(* Logix 5000 project; controller ProyectoAPM Emulate 5570 rev 30.12; software revision 30.00 *)

TASK MainTask (continuous, watchdog 500 ms) : MainProgram

MODULES
   Local : Emulate 5570 (ICP 2, rev 30.12)
      VIRTUAL_OUTPUTS : vendor 1 type 0 code 15 (ICP 4, rev 1.1, Output RPI 50 ms)
      VIRTUAL_INPUTS : vendor 1 type 0 code 15 (ICP 3, rev 1.1, Output RPI 50 ms)
END_MODULES

TYPE HOLE_POSITION :
STRUCT
   X : REAL;
   Y : REAL;
   Z : REAL;
   Z_Hole : REAL;
END_STRUCT
END_TYPE

VAR_GLOBAL   (* controller tags *)
   CNC0_CVB_RUN : BOOL;
   CNC0_CVB_SNR : BOOL;
   DRI0_AXIS_RUN : BOOL;
   DRI0_AXIS_X_AIM_POS : REAL;
   DRI0_AXIS_X_POS : REAL;
   DRI0_AXIS_X_SNR : REAL;
   DRI0_AXIS_Y_AIM_POS : REAL;
   DRI0_AXIS_Y_POS : REAL;
   DRI0_AXIS_Y_SNR : REAL;
   DRI0_AXIS_Z_AIM_POS : REAL;
   DRI0_AXIS_Z_POS : REAL;
   DRI0_AXIS_Z_SNR : REAL;
   DRI0_CVB_RUN : BOOL;
   DRI0_CVB_SNR : BOOL;
   HOLES_PER_TEMPLATE : DINT[4] := ([0] := 20, [1] := 4, [2] := 4, [3] := 4); {constant}
   Hommed : BOOL;
   MOR0_C0_BSW : BOOL;
   MOR0_C0_ESW : BOOL;
   MOR0_C0_VAL : BOOL;
   MOR0_C1_BSW : BOOL;
   MOR0_C1_ESW : BOOL;
   MOR0_C1_VAL : BOOL;
   MOR1_C0_BSW : BOOL;
   MOR1_C0_ESW : BOOL;
   MOR1_C0_VAL : BOOL;
   MOR1_C1_BSW : BOOL;
   MOR1_C1_ESW : BOOL;
   MOR1_C1_VAL : BOOL;
   PAN0_DRI0_CVB_RUN_PB : BOOL;
   PAN0_RST_PB : BOOL;
   PAN0_STP_PB : BOOL;
   PAN0_STT_PB : BOOL;
   PIN0_CVB_RUN : BOOL;
   PIN0_CVB_SNR : BOOL;
   RBT0_CNC0_CVB_RUN : BOOL;
   RBT0_CNC0_CVB_SNR : BOOL;
   RBT0_PIN0_CVB_RUN : BOOL;
   RBT0_PIN0_CVB_SNR : BOOL;
   RBT0_RST_PB : BOOL;
   RBT0_STP_PB : BOOL;
   RBT0_STT_PB : BOOL;
   RBT0_VAL_RUN : BOOL;
   RMT_CNC0_CVB_RUN : BOOL;
   S0_INIT : BOOL;
   S1_CFG : BOOL;
   S2_STBY : BOOL;
   S3_CNC0 : BOOL;
   S3_S0_RUN : BOOL;   // CNC0 Operación Normal de Cinta Transportadora
   S3_S1_STP : BOOL;   // CNC0 Parada de Cinta Transportadora
   S3_S2_STT : BOOL;   // CNC0 Arranque de Cinta Transportadora
   S3_Timer : TIMER := (PRE := 2000);
   S3_TIMER2 : TIMER := (PRE := 10);
   S4_CVB_RQ_ACK : BOOL;
   S4_PIN0 : BOOL;
   S4_S0_RUN : BOOL;   // PIN0 Operación normal de la cinta transportadora con mordazas abiertas
   S4_S1_STP : BOOL;   // PIN0 Parada de Cinta transportadora
   S4_S2_CLE : BOOL;   // PIN0 Cierre de mordazas
   S4_S3_OPN : BOOL;   // PIN0 Apertura de mordazas
   S4_S4_STT : BOOL;   // PIN0 Arranque de cinta transportadora
   S4_Timer0 : TIMER := (PRE := 1000);
   S4_Timer1 : TIMER := (PRE := 2000);
   S4_TIMER2 : TIMER := (PRE := 10);
   S5_COUNTS : INT;
   S5_CURRENT_TEMPLATE : DINT;
   S5_CVB_RQ : BOOL;
   S5_DRI0 : BOOL;
   S5_S0_BYS : BOOL;   // DRI0 Estado de bypass de pasada de primeras piezas
   S5_S1_WAIT_DONE : BOOL;
   S5_S1_WAT : BOOL;   // DRI0 Estato de espera de conteo de primeras piezas
   S5_S1_WAT_END : BOOL;
   S5_S2_RUN : BOOL;   // DRI0 Operación normal de la cinta transportadora con mordazas abiertas
   S5_S3_S0_SBY : BOOL;
   S5_S3_STP : BOOL;   // DRI0 Parada de Cinta transportadora
   S5_S4_CLE : BOOL;   // DRI0 Cierre de mordazas
   S5_S5_DRI : BOOL;   // DRI0 Taladrado
   S5_S5_S0_MOV : BOOL;
   S5_S5_S1_HLE : BOOL;
   S5_S5_S2_UP : BOOL;
   S5_S5_S3_ITR : BOOL;
   S5_S5_S4_EVL : BOOL;
   S5_S5_TIMER0 : TIMER := (PRE := 1000);
   S5_S5_TIMER1 : TIMER := (PRE := 1000);
   S5_S5_TIMER10 : TIMER := (PRE := 1000);
   S5_S5_TIMER11 : TIMER := (PRE := 1000);
   S5_S5_TIMER2 : TIMER := (PRE := 1000);
   S5_S5_TIMER3 : TIMER := (PRE := 1000);
   S5_S5_TIMER4 : TIMER := (PRE := 1000);
   S5_S5_TIMER5 : TIMER := (PRE := 1000);
   S5_S5_TIMER6 : TIMER := (PRE := 1000);
   S5_S5_TIMER7 : TIMER := (PRE := 1000);
   S5_S5_TIMER8 : TIMER := (PRE := 1000);
   S5_S5_TIMER9 : TIMER := (PRE := 1000);
   S5_S6_OPN : BOOL;   // DRI0 Apertura de Mordazas
   S5_S7_STT : BOOL;   // DRI0 Arranque de cinta transportadora durante 2 segundos
   S5_Timer0 : TIMER := (PRE := 2000);
   S5_Timer1 : TIMER := (PRE := 1000);
   S5_Timer2 : TIMER := (PRE := 2000);
   S5_TMP1_IDX : DINT;
   S5_TMP1_INIT : BOOL;
   T0 : BOOL;
   T1 : BOOL;
   T2 : BOOL;
   T3 : BOOL;
   T4 : BOOL;
   T5 : BOOL;
   TEMPLATE1_HOLES : HOLE_POSITION[20] := ([0].X := 14.178, [0].Y := 12.636, [0].Z := 15.692, [0].Z_Hole := 0.692, [1].X := 53.069, [1].Y := 19.708, [1].Z := 15.692, [1].Z_Hole := 0.692, [2].X := 14.178, [2].Y := 177.636, [2].Z := 15.692, [2].Z_Hole := 0.692, [3].X := 14.178, [3].Y := 177.636, [3].Z := 15.692, [3].Z_Hole := 0.692, [4].X := 53.069, [4].Y := 184.708, [4].Z := 15.692, [4].Z_Hole := 0.692, [5].X := 74.282, [5].Y := 205.921, [5].Z := 15.692, [5].Z_Hole := 0.692, [6].X := 14.178, [6].Y := 342.636, [6].Z := 15.692, [6].Z_Hole := 0.692, [7].X := 53.069, [7].Y := 349.708, [7].Z := 15.692, [7].Z_Hole := 0.692, [8].X := 74.282, [8].Y := 370.921, [8].Z := 15.692, [8].Z_Hole := 0.692, [9].X := 14.178, [9].Y := 507.636, [9].Z := 15.692, [9].Z_Hole := 0.692, [10].X := 53.069, [10].Y := 514.708, [10].Z := 15.692, [10].Z_Hole := 0.692, [11].X := 74.282, [11].Y := 535.921, [11].Z := 15.692, [11].Z_Hole := 0.692, [12].X := 134.945, [12].Y := 81.897, [12].Z := 15.692, [12].Z_Hole := 0.692, [13].X := 134.945, [13].Y := 95.897, [13].Z := 15.692, [13].Z_Hole := 0.692, [14].X := 134.156, [14].Y := 440.028, [14].Z := 15.692, [14].Z_Hole := 0.692,
        [15].X := 134.156, [15].Y := 454.028, [15].Z := 15.692, [15].Z_Hole := 0.692, [16].X := 342.588, [16].Y := 142.755, [16].Z := 292.792, [16].Z_Hole := 256.992, [17].X := 342.588, [17].Y := 446.594, [17].Z := 292.792, [17].Z_Hole := 256.992, [18].X := 412.588, [18].Y := 142.755, [18].Z := 292.792, [18].Z_Hole := 256.992, [19].X := 412.588, [19].Y := 446.594, [19].Z := 292.792, [19].Z_Hole := 256.992); {constant}
   TEMPLATE2_HOLES : HOLE_POSITION[4] := ([0].X := 73.196, [0].Y := 300.262, [0].Z := 15.692, [0].Z_Hole := 0.692, [1].X := 225.088, [1].Y := 148.343, [1].Z := 15.692, [1].Z_Hole := 0.692, [2].X := 377.008, [2].Y := 300.262, [2].Z := 15.692, [2].Z_Hole := 0.692, [3].X := 225.088, [3].Y := 452.182, [3].Z := 15.692, [3].Z_Hole := 0.692); {constant}
END_VAR

PROGRAM MainProgram   (* main routine MAIN_GRAFCET *)

ROUTINE MAIN_GRAFCET   (* ladder *)
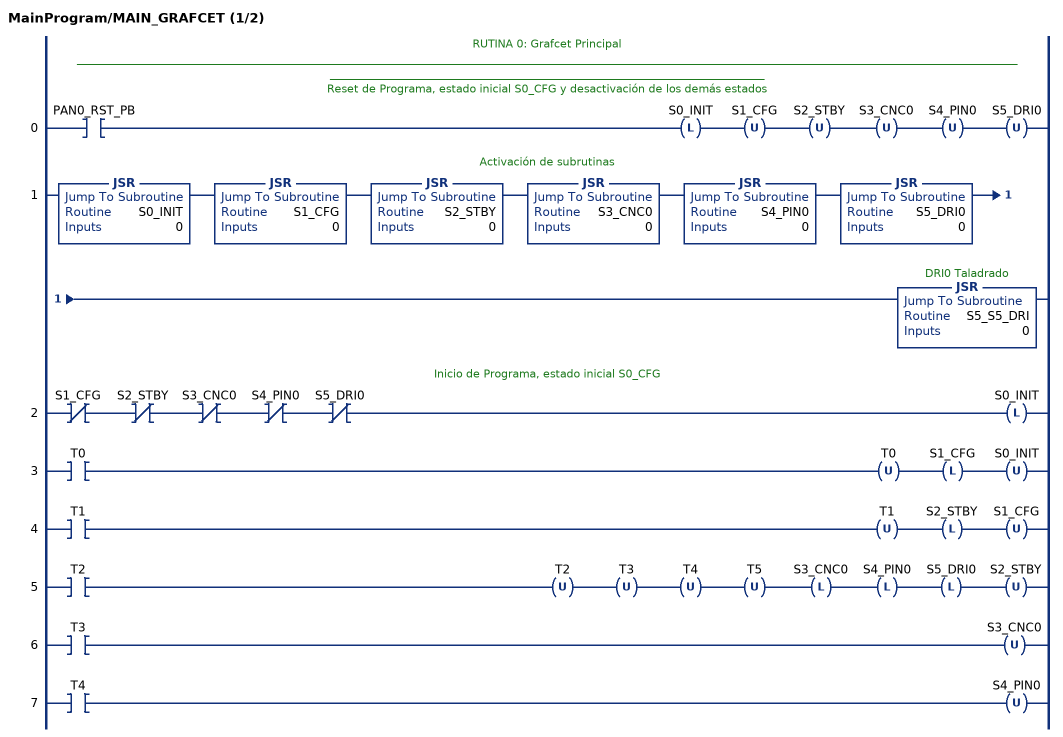
   // RUTINA 0: Grafcet Principal
   // __________________________________________________________________________________________________________________________________________________________________________________________________________________________________________________________
   // Reset de Programa, estado inicial S0_CFG y desactivación de los demás estados
   0: XIC(PAN0_RST_PB)OTL(S0_INIT)OTU(S1_CFG)OTU(S2_STBY)OTU(S3_CNC0)OTU(S4_PIN0)OTU(S5_DRI0);
   // Activación de subrutinas
   1: JSR(S0_INIT,0)JSR(S1_CFG,0)JSR(S2_STBY,0)JSR(S3_CNC0,0)JSR(S4_PIN0,0)JSR(S5_DRI0,0)JSR(S5_S5_DRI,0);
   // Inicio de Programa, estado inicial S0_CFG
   2: XIO(S1_CFG)XIO(S2_STBY)XIO(S3_CNC0)XIO(S4_PIN0)XIO(S5_DRI0)OTL(S0_INIT);
   3: XIC(T0)OTU(T0)OTL(S1_CFG)OTU(S0_INIT);
   4: XIC(T1)OTU(T1)OTL(S2_STBY)OTU(S1_CFG);
   5: XIC(T2)OTU(T2)OTU(T3)OTU(T4)OTU(T5)OTL(S3_CNC0)OTL(S4_PIN0)OTL(S5_DRI0)OTU(S2_STBY);
   6: XIC(T3)OTU(S3_CNC0);
   7: XIC(T4)OTU(S4_PIN0);
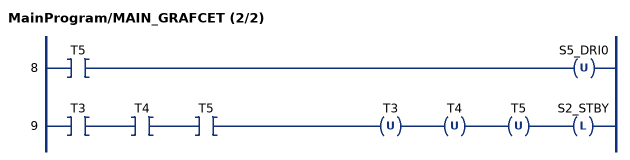
   8: XIC(T5)OTU(S5_DRI0);
   9: XIC(T3)XIC(T4)XIC(T5)OTU(T3)OTU(T4)OTU(T5)OTL(S2_STBY);
END_ROUTINE

ROUTINE S0_INIT   (* ladder *)
// Rutina de inicialización de variables.
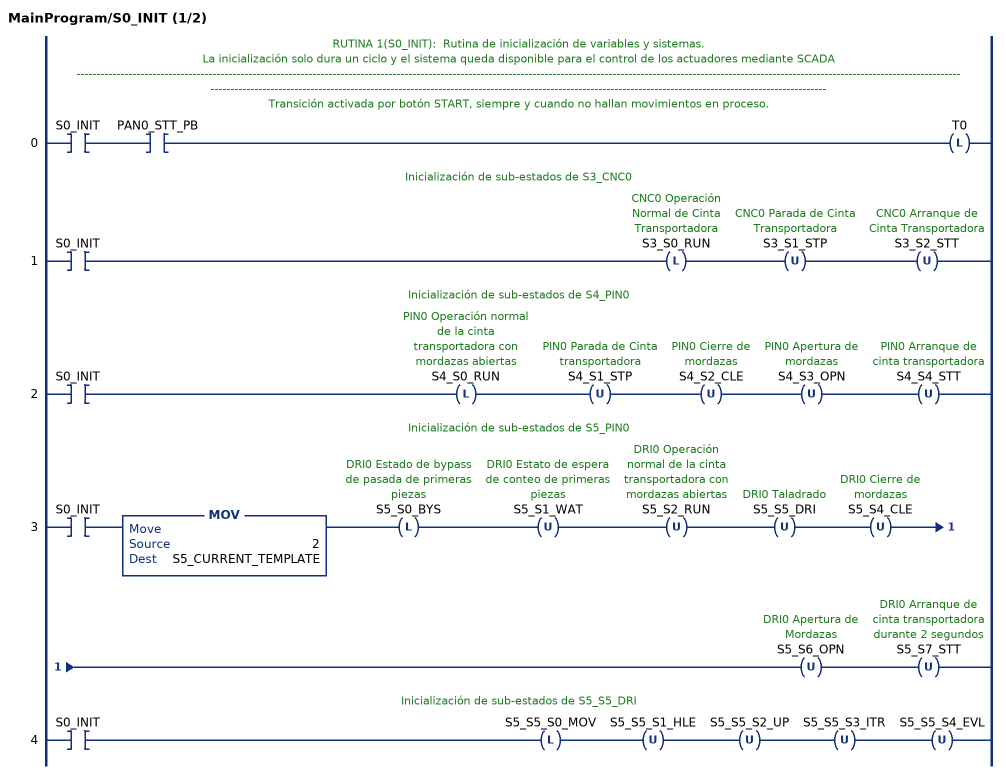
   // RUTINA 1(S0_INIT):  Rutina de inicialización de variables y sistemas.
   // La inicialización solo dura un ciclo y el sistema queda disponible para el control de los actuadores mediante SCADA
   // ---------------------------------------------------------------------------------------------------------------------------------------------------------------------------------------------------------------------------------------------------------------------------------------------------------------------------------------------------------------------------------------
   // Transición activada por botón START, siempre y cuando no hallan movimientos en proceso.
   0: XIC(S0_INIT)XIC(PAN0_STT_PB)OTL(T0);
   // Inicialización de sub-estados de S3_CNC0
   1: XIC(S0_INIT)OTL(S3_S0_RUN)OTU(S3_S1_STP)OTU(S3_S2_STT);
   // Inicialización de sub-estados de S4_PIN0
   2: XIC(S0_INIT)OTL(S4_S0_RUN)OTU(S4_S1_STP)OTU(S4_S2_CLE)OTU(S4_S3_OPN)OTU(S4_S4_STT);
   // Inicialización de sub-estados de S5_PIN0
   3: XIC(S0_INIT)MOV(2,S5_CURRENT_TEMPLATE)OTL(S5_S0_BYS)OTU(S5_S1_WAT)OTU(S5_S2_RUN)OTU(S5_S5_DRI)OTU(S5_S4_CLE)OTU(S5_S6_OPN)OTU(S5_S7_STT);
   // Inicialización de sub-estados de S5_S5_DRI
   4: XIC(S0_INIT)OTL(S5_S5_S0_MOV)OTU(S5_S5_S1_HLE)OTU(S5_S5_S2_UP)OTU(S5_S5_S3_ITR)OTU(S5_S5_S4_EVL);
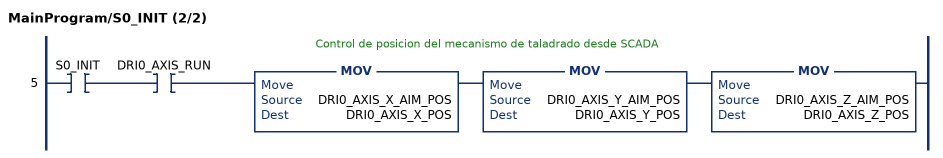
   // Control de posicion del mecanismo de taladrado desde SCADA
   5: XIC(S0_INIT)XIC(DRI0_AXIS_RUN)MOV(DRI0_AXIS_X_AIM_POS,DRI0_AXIS_X_POS)MOV(DRI0_AXIS_Y_AIM_POS,DRI0_AXIS_Y_POS)MOV(DRI0_AXIS_Z_AIM_POS,DRI0_AXIS_Z_POS);
END_ROUTINE

ROUTINE S1_CFG   (* ladder *)
// Homing de los actuadores
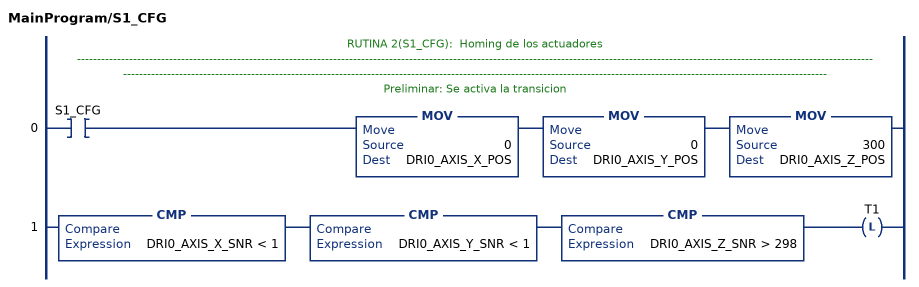
   // RUTINA 2(S1_CFG):  Homing de los actuadores
   // ---------------------------------------------------------------------------------------------------------------------------------------------------------------------------------------------------------------------------------------------------------------------------------------------------------------------------------------------------------------------------------------
   // Preliminar: Se activa la transicion
   0: XIC(S1_CFG)MOV(0,DRI0_AXIS_X_POS)MOV(0,DRI0_AXIS_Y_POS)MOV(300,DRI0_AXIS_Z_POS);
   1: CMP(DRI0_AXIS_X_SNR < 1)CMP(DRI0_AXIS_Y_SNR < 1)CMP(DRI0_AXIS_Z_SNR > 298)OTL(T1);
END_ROUTINE

ROUTINE S2_STBY   (* ladder *)
// Modo de espera/Pausa
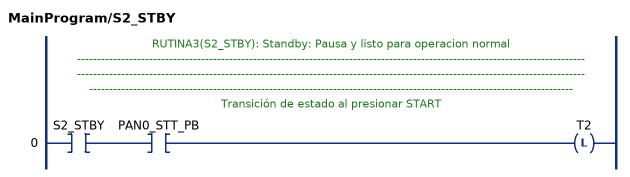
   // RUTINA3(S2_STBY): Standby: Pausa y listo para operacion normal
   // ---------------------------------------------------------------------------------------------------------------------------------------------------------------------------------------------------------------------------------------------------------------------------------------------------------------------------------------------------------------------------------------
   // Transición de estado al presionar START
   0: XIC(S2_STBY)XIC(PAN0_STT_PB)OTL(T2);
END_ROUTINE

ROUTINE S3_CNC0   (* ladder *)
// Operación normal de los elementos asociados a la celda de la fresadora CNC
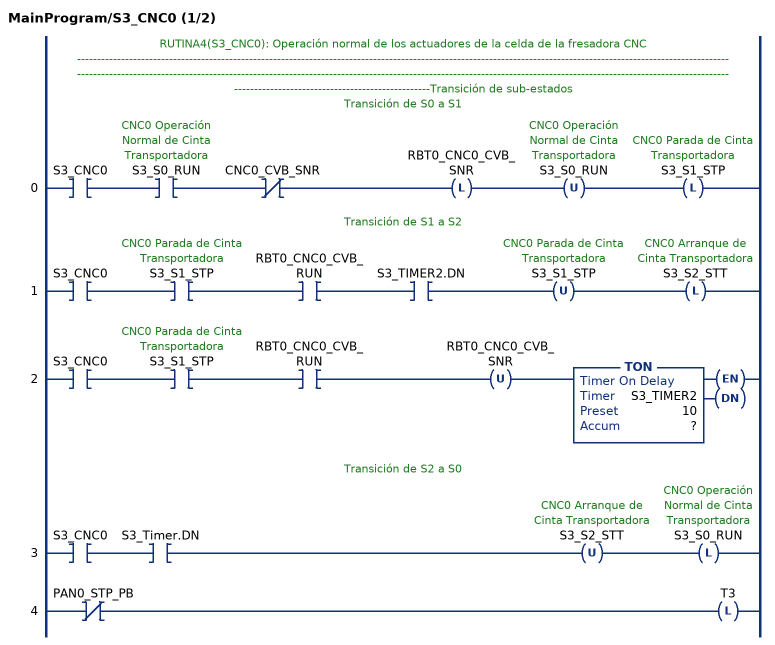
   // RUTINA4(S3_CNC0): Operación normal de los actuadores de la celda de la fresadora CNC
   // ---------------------------------------------------------------------------------------------------------------------------------------------------------------------------------------------------------------------------------------------------------------------------------------------------------------------------------------------------------------------------------------Transición de sub-estados
   // Transición de S0 a S1
   0: XIC(S3_CNC0)XIC(S3_S0_RUN)XIO(CNC0_CVB_SNR)OTL(RBT0_CNC0_CVB_SNR)OTU(S3_S0_RUN)OTL(S3_S1_STP);
   // Transición de S1 a S2
   1: XIC(S3_CNC0)XIC(S3_S1_STP)XIC(RBT0_CNC0_CVB_RUN)XIC(S3_TIMER2.DN)OTU(S3_S1_STP)OTL(S3_S2_STT);
   2: XIC(S3_CNC0)XIC(S3_S1_STP)XIC(RBT0_CNC0_CVB_RUN)OTU(RBT0_CNC0_CVB_SNR)TON(S3_TIMER2,?,?);
   // Transición de S2 a S0
   3: XIC(S3_CNC0)XIC(S3_Timer.DN)OTU(S3_S2_STT)OTL(S3_S0_RUN);
   4: XIO(PAN0_STP_PB)OTL(T3);
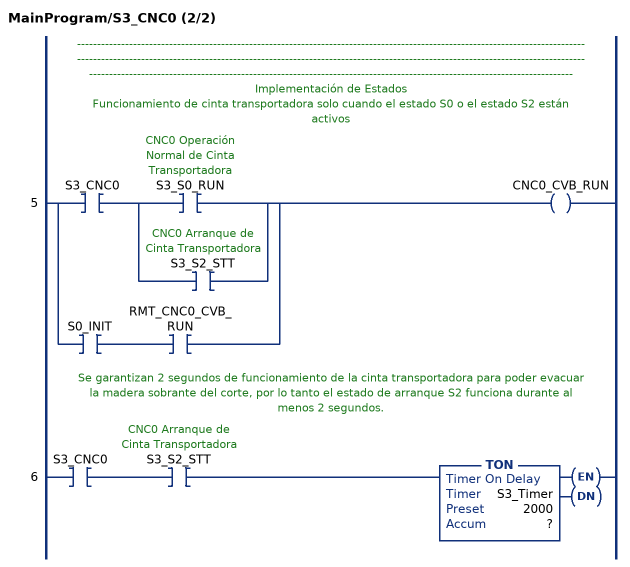
   // --------------------------------------------------------------------------------------------------------------------------------------------------------------------------------------------------------------------------------------------------------------------------------------------------------------------------------------------------------------------------------------- Implementación de Estados
   // Funcionamiento de cinta transportadora solo cuando el estado S0 o el estado S2 están activos
   5: [XIC(S3_CNC0) [XIC(S3_S0_RUN) ,XIC(S3_S2_STT) ] ,XIC(S0_INIT) XIC(RMT_CNC0_CVB_RUN) ]OTE(CNC0_CVB_RUN);
   // Se garantizan 2 segundos de funcionamiento de la cinta transportadora para poder evacuar la madera sobrante del corte, por lo tanto el estado de arranque S2 funciona durante al menos 2 segundos.
   6: XIC(S3_CNC0)XIC(S3_S2_STT)TON(S3_Timer,?,?);
END_ROUTINE

ROUTINE S4_PIN0   (* ladder *)
// Operación normal de los actuadores de la celda de intercambio de partes
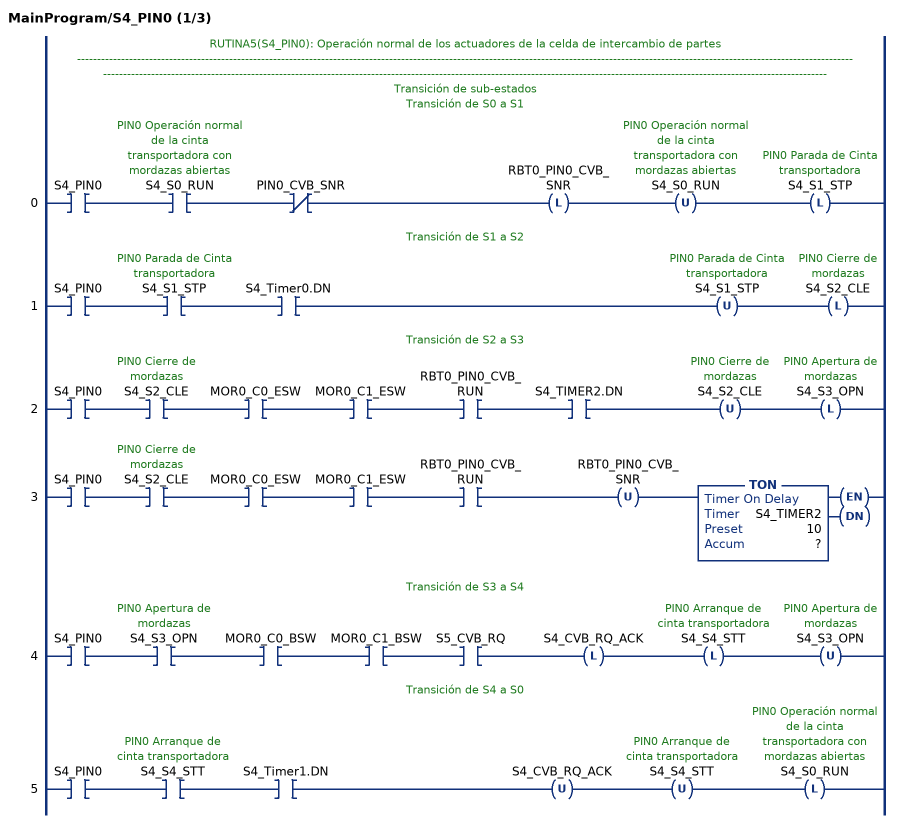
   // RUTINA5(S4_PIN0): Operación normal de los actuadores de la celda de intercambio de partes
   // ---------------------------------------------------------------------------------------------------------------------------------------------------------------------------------------------------------------------------------------------------------------------------------------------------------------------------------------------------------------------------------------Transición de sub-estados
   // Transición de S0 a S1
   0: XIC(S4_PIN0)XIC(S4_S0_RUN)XIO(PIN0_CVB_SNR)OTL(RBT0_PIN0_CVB_SNR)OTU(S4_S0_RUN)OTL(S4_S1_STP);
   // Transición de S1 a S2
   1: XIC(S4_PIN0)XIC(S4_S1_STP)XIC(S4_Timer0.DN)OTU(S4_S1_STP)OTL(S4_S2_CLE);
   // Transición de S2 a S3
   2: XIC(S4_PIN0)XIC(S4_S2_CLE)XIC(MOR0_C0_ESW)XIC(MOR0_C1_ESW)XIC(RBT0_PIN0_CVB_RUN)XIC(S4_TIMER2.DN)OTU(S4_S2_CLE)OTL(S4_S3_OPN);
   3: XIC(S4_PIN0)XIC(S4_S2_CLE)XIC(MOR0_C0_ESW)XIC(MOR0_C1_ESW)XIC(RBT0_PIN0_CVB_RUN)OTU(RBT0_PIN0_CVB_SNR)TON(S4_TIMER2,?,?);
   // Transición de S3 a S4
   4: XIC(S4_PIN0)XIC(S4_S3_OPN)XIC(MOR0_C0_BSW)XIC(MOR0_C1_BSW)XIC(S5_CVB_RQ)OTL(S4_CVB_RQ_ACK)OTL(S4_S4_STT)OTU(S4_S3_OPN);
   // Transición de S4 a S0
   5: XIC(S4_PIN0)XIC(S4_S4_STT)XIC(S4_Timer1.DN)OTU(S4_CVB_RQ_ACK)OTU(S4_S4_STT)OTL(S4_S0_RUN);
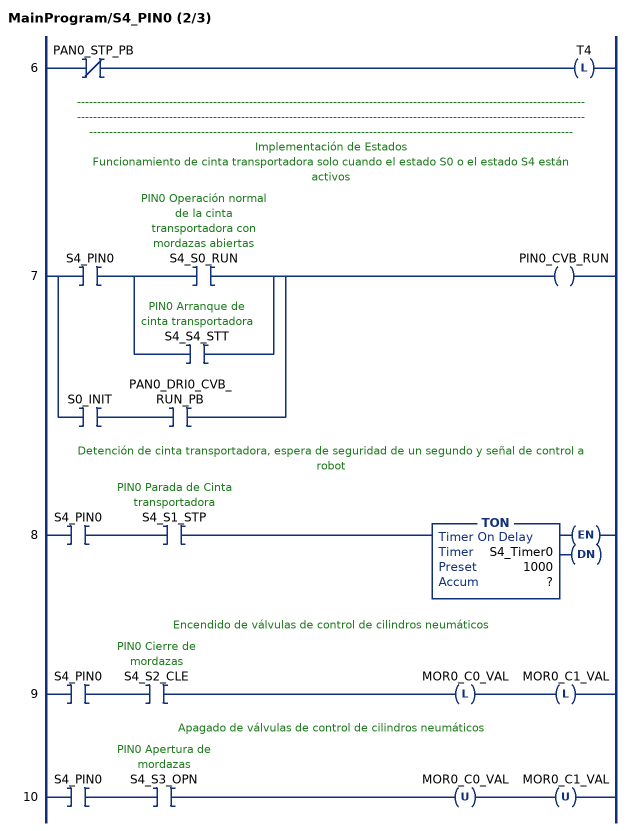
   6: XIO(PAN0_STP_PB)OTL(T4);
   // --------------------------------------------------------------------------------------------------------------------------------------------------------------------------------------------------------------------------------------------------------------------------------------------------------------------------------------------------------------------------------------- Implementación de Estados
   // Funcionamiento de cinta transportadora solo cuando el estado S0 o el estado S4 están activos
   7: [XIC(S4_PIN0) [XIC(S4_S0_RUN) ,XIC(S4_S4_STT) ] ,XIC(S0_INIT) XIC(PAN0_DRI0_CVB_RUN_PB) ]OTE(PIN0_CVB_RUN);
   // Detención de cinta transportadora, espera de seguridad de un segundo y señal de control a robot
   8: XIC(S4_PIN0)XIC(S4_S1_STP)TON(S4_Timer0,?,?);
   // Encendido de válvulas de control de cilindros neumáticos
   9: XIC(S4_PIN0)XIC(S4_S2_CLE)OTL(MOR0_C0_VAL)OTL(MOR0_C1_VAL);
   // Apagado de válvulas de control de cilindros neumáticos
   10: XIC(S4_PIN0)XIC(S4_S3_OPN)OTU(MOR0_C0_VAL)OTU(MOR0_C1_VAL);
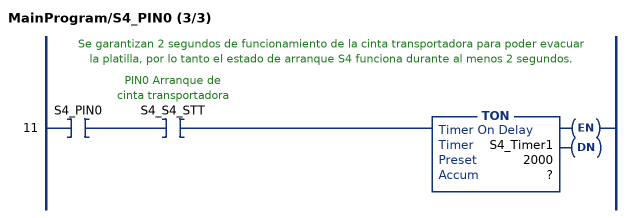
   // Se garantizan 2 segundos de funcionamiento de la cinta transportadora para poder evacuar la platilla, por lo tanto el estado de arranque S4 funciona durante al menos 2 segundos.
   11: XIC(S4_PIN0)XIC(S4_S4_STT)TON(S4_Timer1,?,?);
END_ROUTINE

ROUTINE S5_DRI0   (* ladder *)
// Operación normal de los actuadores de la celda de taladrado
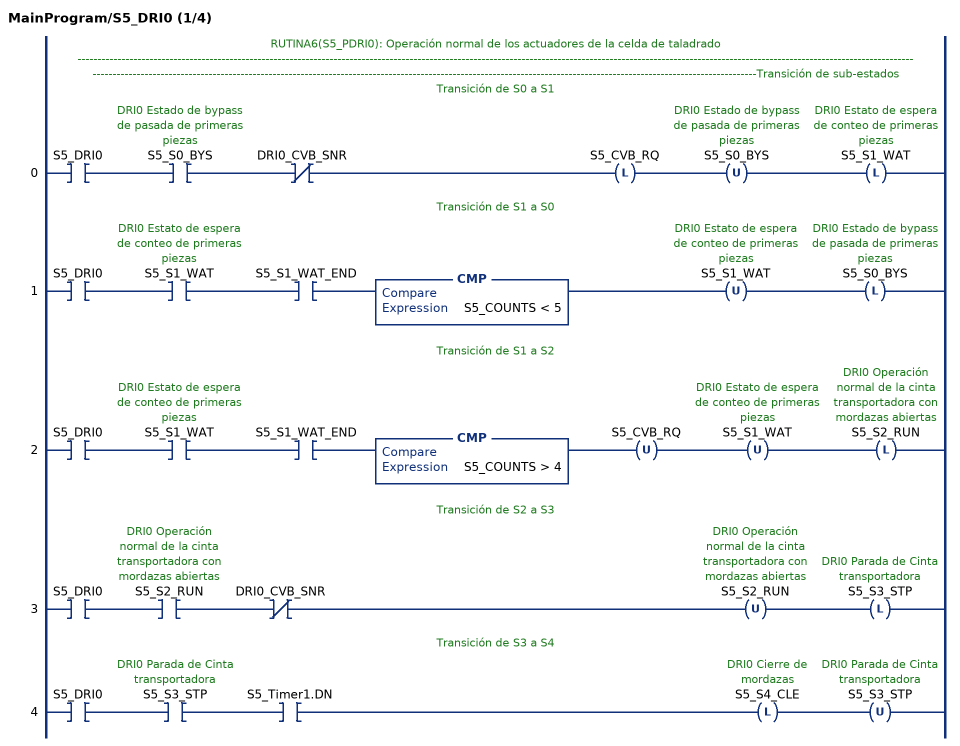
   // RUTINA6(S5_PDRI0): Operación normal de los actuadores de la celda de taladrado
   // ---------------------------------------------------------------------------------------------------------------------------------------------------------------------------------------------------------------------------------------------------------------------------------------------------------------------------------------------------------------------------------------Transición de sub-estados
   // Transición de S0 a S1
   0: XIC(S5_DRI0)XIC(S5_S0_BYS)XIO(DRI0_CVB_SNR)OTL(S5_CVB_RQ)OTU(S5_S0_BYS)OTL(S5_S1_WAT);
   // Transición de S1 a S0
   1: XIC(S5_DRI0)XIC(S5_S1_WAT)XIC(S5_S1_WAT_END)CMP(S5_COUNTS < 5)OTU(S5_S1_WAT)OTL(S5_S0_BYS);
   // Transición de S1 a S2
   2: XIC(S5_DRI0)XIC(S5_S1_WAT)XIC(S5_S1_WAT_END)CMP(S5_COUNTS > 4)OTU(S5_CVB_RQ)OTU(S5_S1_WAT)OTL(S5_S2_RUN);
   // Transición de S2 a S3
   3: XIC(S5_DRI0)XIC(S5_S2_RUN)XIO(DRI0_CVB_SNR)OTU(S5_S2_RUN)OTL(S5_S3_STP);
   // Transición de S3 a S4
   4: XIC(S5_DRI0)XIC(S5_S3_STP)XIC(S5_Timer1.DN)OTL(S5_S4_CLE)OTU(S5_S3_STP);
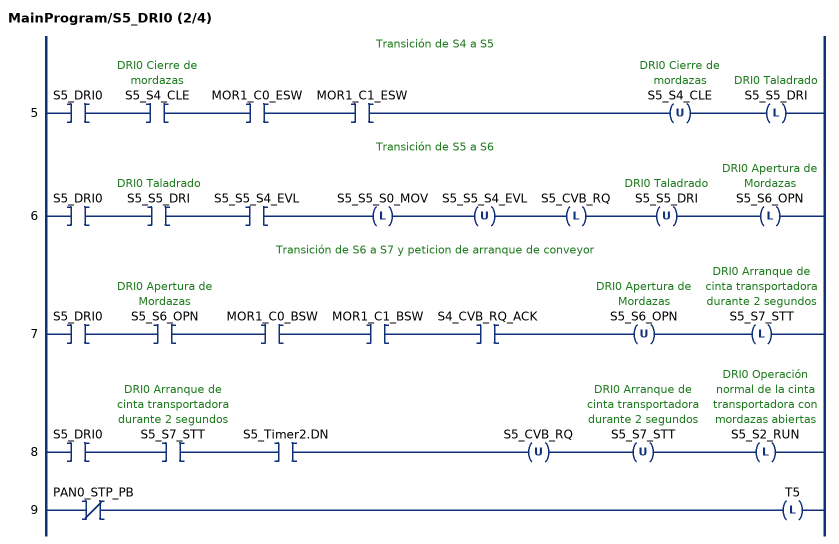
   // Transición de S4 a S5
   5: XIC(S5_DRI0)XIC(S5_S4_CLE)XIC(MOR1_C0_ESW)XIC(MOR1_C1_ESW)OTU(S5_S4_CLE)OTL(S5_S5_DRI);
   // Transición de S5 a S6
   6: XIC(S5_DRI0)XIC(S5_S5_DRI)XIC(S5_S5_S4_EVL)OTL(S5_S5_S0_MOV)OTU(S5_S5_S4_EVL)OTL(S5_CVB_RQ)OTU(S5_S5_DRI)OTL(S5_S6_OPN);
   // Transición de S6 a S7 y peticion de arranque de conveyor
   7: XIC(S5_DRI0)XIC(S5_S6_OPN)XIC(MOR1_C0_BSW)XIC(MOR1_C1_BSW)XIC(S4_CVB_RQ_ACK)OTU(S5_S6_OPN)OTL(S5_S7_STT);
   8: XIC(S5_DRI0)XIC(S5_S7_STT)XIC(S5_Timer2.DN)OTU(S5_CVB_RQ)OTU(S5_S7_STT)OTL(S5_S2_RUN);
   9: XIO(PAN0_STP_PB)OTL(T5);
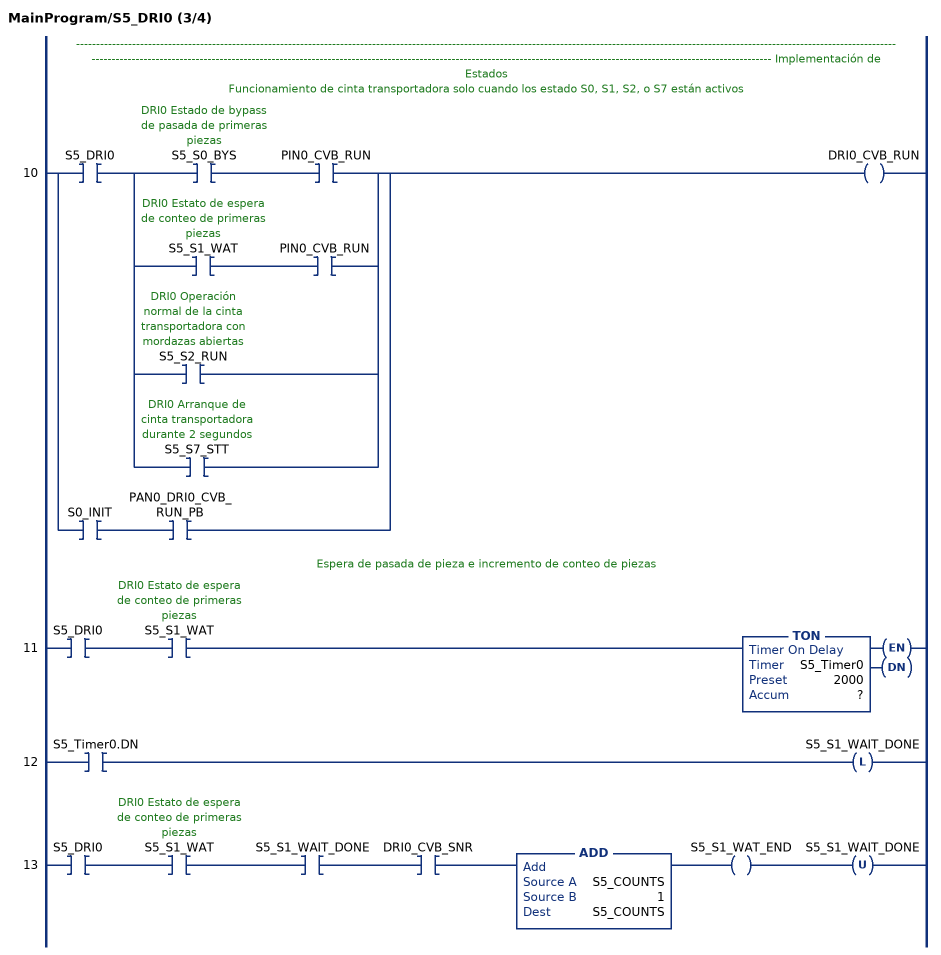
   // --------------------------------------------------------------------------------------------------------------------------------------------------------------------------------------------------------------------------------------------------------------------------------------------------------------------------------------------------------------------------------------- Implementación de Estados
   // Funcionamiento de cinta transportadora solo cuando los estado S0, S1, S2, o S7 están activos
   10: [XIC(S5_DRI0) [XIC(S5_S0_BYS) XIC(PIN0_CVB_RUN) ,[XIC(S5_S1_WAT) XIC(PIN0_CVB_RUN) ,[XIC(S5_S2_RUN) ,XIC(S5_S7_STT) ] ] ] ,XIC(S0_INIT) XIC(PAN0_DRI0_CVB_RUN_PB) ]OTE(DRI0_CVB_RUN);
   // Espera de pasada de pieza e incremento de conteo de piezas
   11: XIC(S5_DRI0)XIC(S5_S1_WAT)TON(S5_Timer0,?,?);
   12: XIC(S5_Timer0.DN)OTL(S5_S1_WAIT_DONE);
   13: XIC(S5_DRI0)XIC(S5_S1_WAT)XIC(S5_S1_WAIT_DONE)XIC(DRI0_CVB_SNR)ADD(S5_COUNTS,1,S5_COUNTS)OTE(S5_S1_WAT_END)OTU(S5_S1_WAIT_DONE);
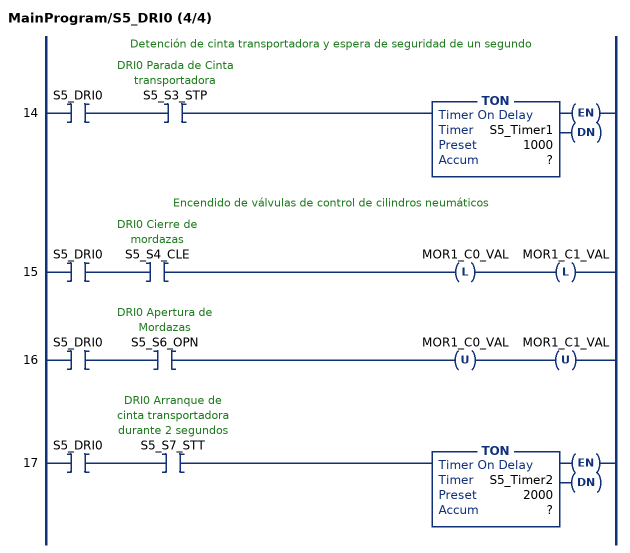
   // Detención de cinta transportadora y espera de seguridad de un segundo
   14: XIC(S5_DRI0)XIC(S5_S3_STP)TON(S5_Timer1,?,?);
   // Encendido de válvulas de control de cilindros neumáticos
   15: XIC(S5_DRI0)XIC(S5_S4_CLE)OTL(MOR1_C0_VAL)OTL(MOR1_C1_VAL);
   16: XIC(S5_DRI0)XIC(S5_S6_OPN)OTU(MOR1_C0_VAL)OTU(MOR1_C1_VAL);
   17: XIC(S5_DRI0)XIC(S5_S7_STT)TON(S5_Timer2,?,?);
END_ROUTINE

ROUTINE S5_S5_DRI   (* ladder *)
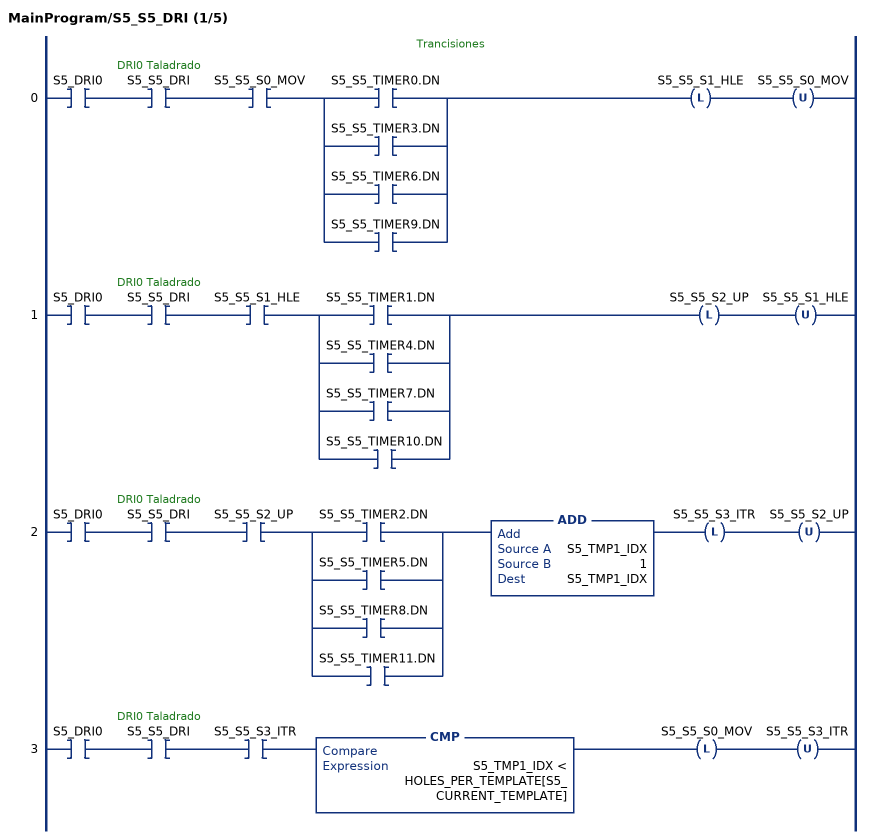
   // Trancisiones
   0: XIC(S5_DRI0)XIC(S5_S5_DRI)XIC(S5_S5_S0_MOV)[XIC(S5_S5_TIMER0.DN) ,[XIC(S5_S5_TIMER3.DN) ,[XIC(S5_S5_TIMER6.DN) ,XIC(S5_S5_TIMER9.DN) ] ] ]OTL(S5_S5_S1_HLE)OTU(S5_S5_S0_MOV);
   1: XIC(S5_DRI0)XIC(S5_S5_DRI)XIC(S5_S5_S1_HLE)[XIC(S5_S5_TIMER1.DN) ,[XIC(S5_S5_TIMER4.DN) ,[XIC(S5_S5_TIMER7.DN) ,XIC(S5_S5_TIMER10.DN) ] ] ]OTL(S5_S5_S2_UP)OTU(S5_S5_S1_HLE);
   2: XIC(S5_DRI0)XIC(S5_S5_DRI)XIC(S5_S5_S2_UP)[XIC(S5_S5_TIMER2.DN) ,[XIC(S5_S5_TIMER5.DN) ,[XIC(S5_S5_TIMER8.DN) ,XIC(S5_S5_TIMER11.DN) ] ] ]ADD(S5_TMP1_IDX,1,S5_TMP1_IDX)OTL(S5_S5_S3_ITR)OTU(S5_S5_S2_UP);
   3: XIC(S5_DRI0)XIC(S5_S5_DRI)XIC(S5_S5_S3_ITR)CMP(S5_TMP1_IDX < HOLES_PER_TEMPLATE[S5_CURRENT_TEMPLATE])OTL(S5_S5_S0_MOV)OTU(S5_S5_S3_ITR);
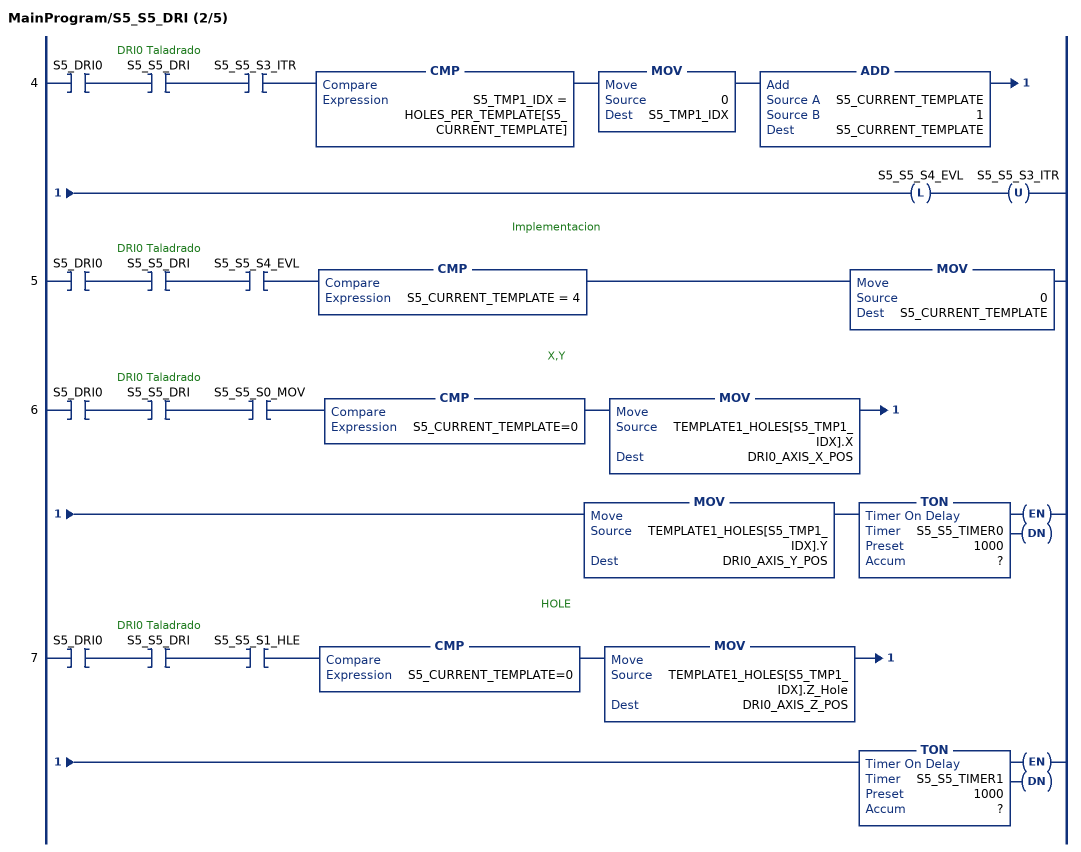
   4: XIC(S5_DRI0)XIC(S5_S5_DRI)XIC(S5_S5_S3_ITR)CMP(S5_TMP1_IDX = HOLES_PER_TEMPLATE[S5_CURRENT_TEMPLATE])MOV(0,S5_TMP1_IDX)ADD(S5_CURRENT_TEMPLATE,1,S5_CURRENT_TEMPLATE)OTL(S5_S5_S4_EVL)OTU(S5_S5_S3_ITR);
   // Implementacion
   5: XIC(S5_DRI0)XIC(S5_S5_DRI)XIC(S5_S5_S4_EVL)CMP(S5_CURRENT_TEMPLATE = 4)MOV(0,S5_CURRENT_TEMPLATE);
   // X,Y
   6: XIC(S5_DRI0)XIC(S5_S5_DRI)XIC(S5_S5_S0_MOV)CMP(S5_CURRENT_TEMPLATE=0)MOV(TEMPLATE1_HOLES[S5_TMP1_IDX].X,DRI0_AXIS_X_POS)MOV(TEMPLATE1_HOLES[S5_TMP1_IDX].Y,DRI0_AXIS_Y_POS)TON(S5_S5_TIMER0,?,?);
   // HOLE
   7: XIC(S5_DRI0)XIC(S5_S5_DRI)XIC(S5_S5_S1_HLE)CMP(S5_CURRENT_TEMPLATE=0)MOV(TEMPLATE1_HOLES[S5_TMP1_IDX].Z_Hole,DRI0_AXIS_Z_POS)TON(S5_S5_TIMER1,?,?);
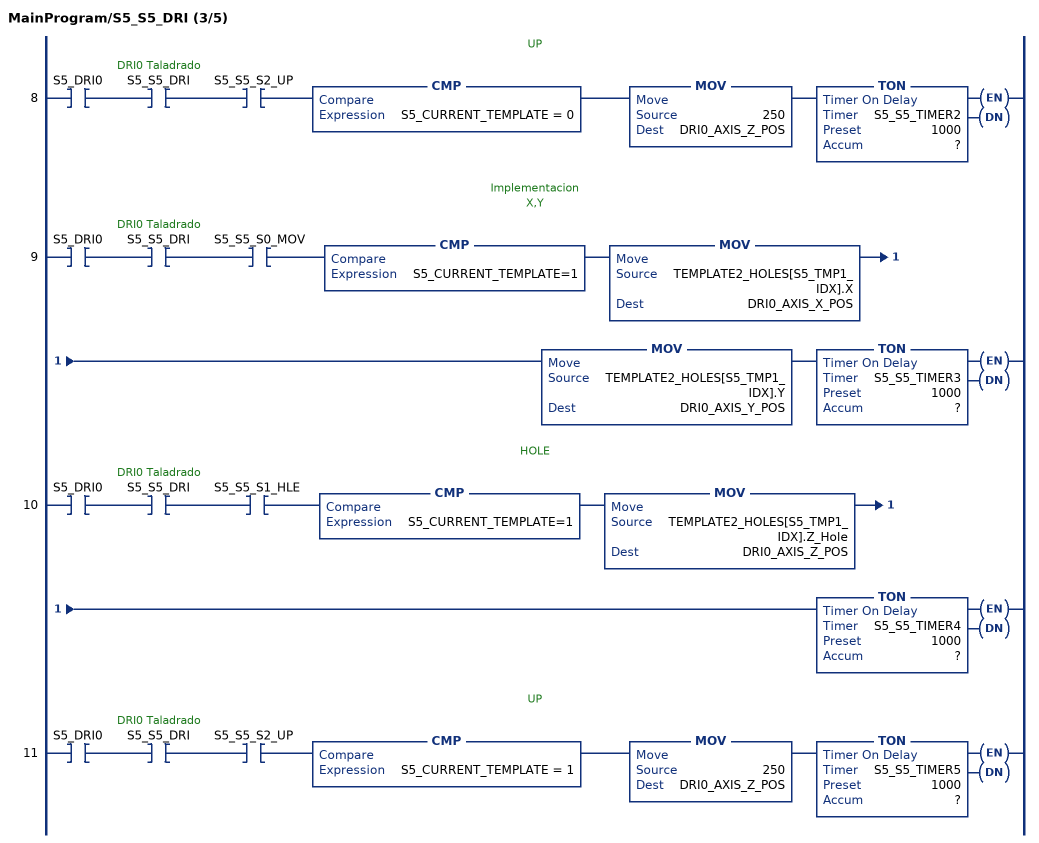
   // UP
   8: XIC(S5_DRI0)XIC(S5_S5_DRI)XIC(S5_S5_S2_UP)CMP(S5_CURRENT_TEMPLATE = 0)MOV(250,DRI0_AXIS_Z_POS)TON(S5_S5_TIMER2,?,?);
   // Implementacion
   // X,Y
   9: XIC(S5_DRI0)XIC(S5_S5_DRI)XIC(S5_S5_S0_MOV)CMP(S5_CURRENT_TEMPLATE=1)MOV(TEMPLATE2_HOLES[S5_TMP1_IDX].X,DRI0_AXIS_X_POS)MOV(TEMPLATE2_HOLES[S5_TMP1_IDX].Y,DRI0_AXIS_Y_POS)TON(S5_S5_TIMER3,?,?);
   // HOLE
   10: XIC(S5_DRI0)XIC(S5_S5_DRI)XIC(S5_S5_S1_HLE)CMP(S5_CURRENT_TEMPLATE=1)MOV(TEMPLATE2_HOLES[S5_TMP1_IDX].Z_Hole,DRI0_AXIS_Z_POS)TON(S5_S5_TIMER4,?,?);
   // UP
   11: XIC(S5_DRI0)XIC(S5_S5_DRI)XIC(S5_S5_S2_UP)CMP(S5_CURRENT_TEMPLATE = 1)MOV(250,DRI0_AXIS_Z_POS)TON(S5_S5_TIMER5,?,?);
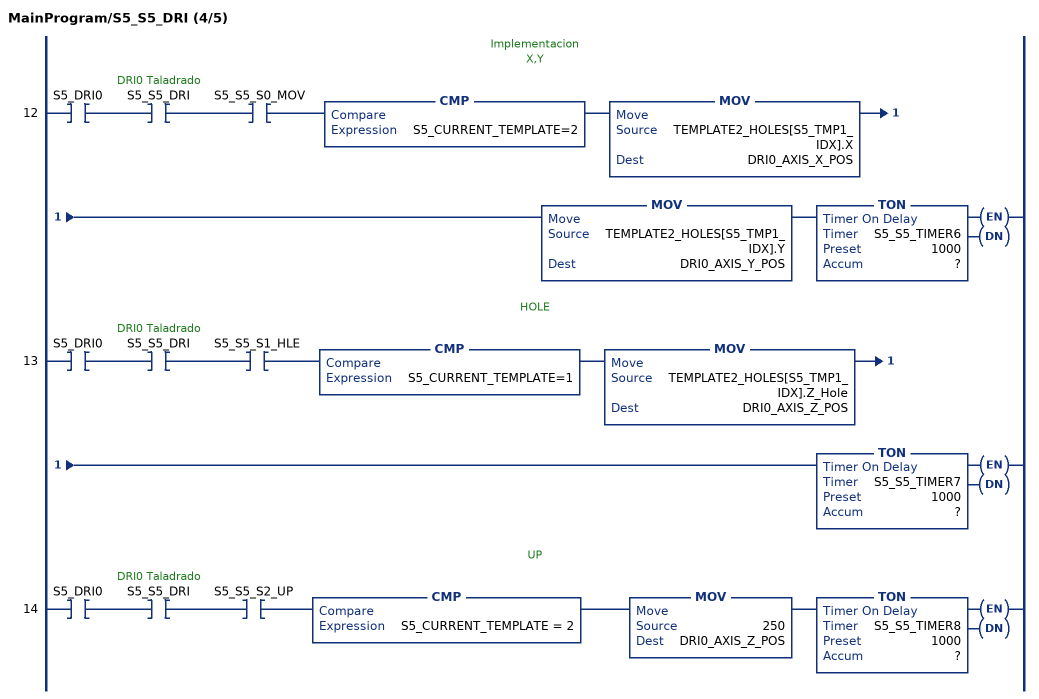
   // Implementacion
   // X,Y
   12: XIC(S5_DRI0)XIC(S5_S5_DRI)XIC(S5_S5_S0_MOV)CMP(S5_CURRENT_TEMPLATE=2)MOV(TEMPLATE2_HOLES[S5_TMP1_IDX].X,DRI0_AXIS_X_POS)MOV(TEMPLATE2_HOLES[S5_TMP1_IDX].Y,DRI0_AXIS_Y_POS)TON(S5_S5_TIMER6,?,?);
   // HOLE
   13: XIC(S5_DRI0)XIC(S5_S5_DRI)XIC(S5_S5_S1_HLE)CMP(S5_CURRENT_TEMPLATE=1)MOV(TEMPLATE2_HOLES[S5_TMP1_IDX].Z_Hole,DRI0_AXIS_Z_POS)TON(S5_S5_TIMER7,?,?);
   // UP
   14: XIC(S5_DRI0)XIC(S5_S5_DRI)XIC(S5_S5_S2_UP)CMP(S5_CURRENT_TEMPLATE = 2)MOV(250,DRI0_AXIS_Z_POS)TON(S5_S5_TIMER8,?,?);
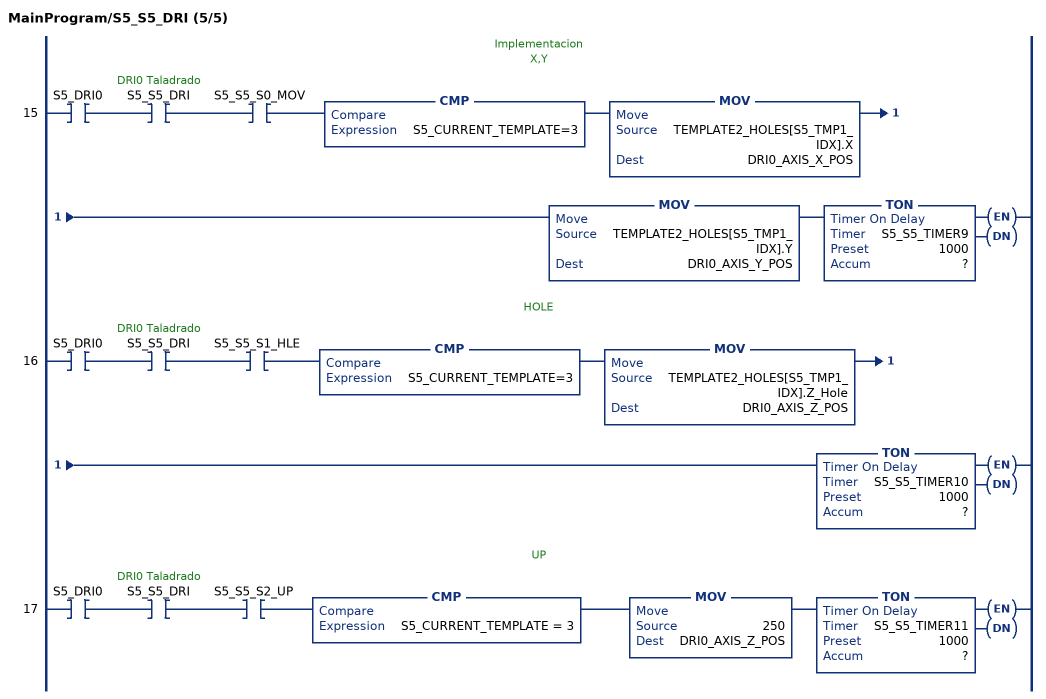
   // Implementacion
   // X,Y
   15: XIC(S5_DRI0)XIC(S5_S5_DRI)XIC(S5_S5_S0_MOV)CMP(S5_CURRENT_TEMPLATE=3)MOV(TEMPLATE2_HOLES[S5_TMP1_IDX].X,DRI0_AXIS_X_POS)MOV(TEMPLATE2_HOLES[S5_TMP1_IDX].Y,DRI0_AXIS_Y_POS)TON(S5_S5_TIMER9,?,?);
   // HOLE
   16: XIC(S5_DRI0)XIC(S5_S5_DRI)XIC(S5_S5_S1_HLE)CMP(S5_CURRENT_TEMPLATE=3)MOV(TEMPLATE2_HOLES[S5_TMP1_IDX].Z_Hole,DRI0_AXIS_Z_POS)TON(S5_S5_TIMER10,?,?);
   // UP
   17: XIC(S5_DRI0)XIC(S5_S5_DRI)XIC(S5_S5_S2_UP)CMP(S5_CURRENT_TEMPLATE = 3)MOV(250,DRI0_AXIS_Z_POS)TON(S5_S5_TIMER11,?,?);
END_ROUTINE
END_PROGRAM
